PROGRAM PRG_ST1K4_TEST
VAR
	fbMotion1: FB_MotionStage;
END_VAR

// M14, Axis 14
Main.M14.nEnableMode	:= ENUM_StageEnableMode.DURING_MOTION;
Main.M14.bHardwareEnable:= TRUE;
Main.M14.bPowerSelf := TRUE;
Main.M14.nBrakeMode := ENUM_StageBrakeMode.IF_ENABLED;
fbMotion1(stMotionStage:=Main.M14);

END_PROGRAM

(* stored: Version 1.1.0.1, ProductVersion 3.1.4022.18
   POU PRG_ST1K4_TEST: Id {75fb9ec1-c09f-44b1-93e4-582e1bc13e2e}, SpecialFunc None *)
